{attribute 'hide_all_locals' := ''}
{attribute 'FBVisuCreator' := ''}
{attribute 'FBVisuCreatorPrefix' := 'RET_VISU_'}
FUNCTION_BLOCK PT2s
VAR_INPUT
	{attribute 'FBVisuCreatorFormatString' := '%1.3f'}
	fX: REAL;
	{attribute 'FBVisuCreatorFormatString' := '%1.3f'}
	fK: REAL;
	{attribute 'FBVisuCreatorFormatString' := '%1.3f'}
	fZeta: REAL;
	{attribute 'FBVisuCreatorFormatString' := '%1.3f'}
	fOmega: REAL;
	{attribute 'FBVisuCreatorBoolColor' := 'Red'}
	bReset: BOOL;
END_VAR
VAR_OUTPUT
	{attribute 'FBVisuCreatorFormatString' := '%1.3f'}
	fY: REAL;
END_VAR
VAR
	{attribute 'hide'}
	fXX: REAL;
	{attribute 'hide'}
	fDx: REAL;
	{attribute 'hide'}
	fDy: REAL;
END_VAR

fDy := RET_COMMON.fDt*fOmega*fXX;
fDx := RET_COMMON.fDt*fOmega*(fK*fX - fY - 2*fZeta*fXX);
fXX := fXX + fDx;
fY := fY + fDy;

IF bReset THEN
	reset();
END_IF

ACTION reset:
fXX := 0.0;
fY := 0.0;
END_ACTION

END_FUNCTION_BLOCK

(* stored: Version 1.1.0.1, ProductVersion 3.1.4024.12
   POU PT2s: Id {6a40dc06-492f-41dd-a803-d5d2799b6bff}, SpecialFunc None
   Action reset: Id {2682f867-340b-4886-ab96-4b023d721e7b} *)
